// SIMATIC S7-200 project (STEP 7-Micro/WIN), CPU 224XP REL 02.01

SYMBOL_TABLE USER1
start            I0.0
stop_btn         I0.1
x1               Q0.0
v1               Q0.1
d1               Q0.2
x2               Q0.3
v2               Q0.4
d2               Q0.5
END_SYMBOL_TABLE

ORGANIZATION_BLOCK MAIN:OB1
TITLE=PROGRAM COMMENTS
BEGIN
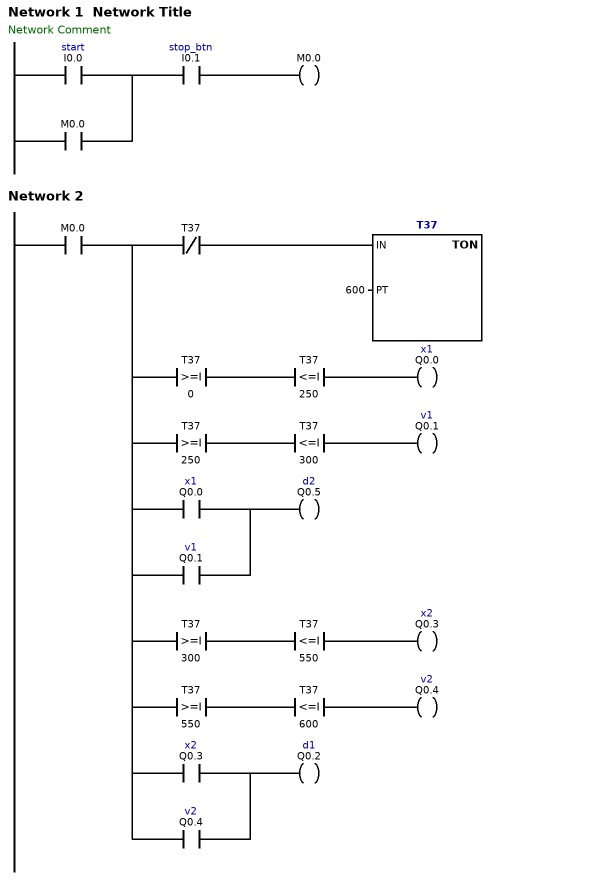
Network 1 // Network Title
// Network Comment
LD     start:I0.0
O      M0.0
A      stop_btn:I0.1
=      M0.0
Network 2
LD     M0.0
LPS
AN     T37
TON    T37, 600
LRD
AW>=   T37, 0
AW<=   T37, 250
=      x1:Q0.0
LRD
AW>=   T37, 250
AW<=   T37, 300
=      v1:Q0.1
LRD
LD     x1:Q0.0
O      v1:Q0.1
ALD
=      d2:Q0.5
LRD
LPS
AW>=   T37, 300
AW<=   T37, 550
=      x2:Q0.3
LPP
AW>=   T37, 550
AW<=   T37, 600
=      v2:Q0.4
LPP
LD     x2:Q0.3
O      v2:Q0.4
ALD
=      d1:Q0.2
END_ORGANIZATION_BLOCK
